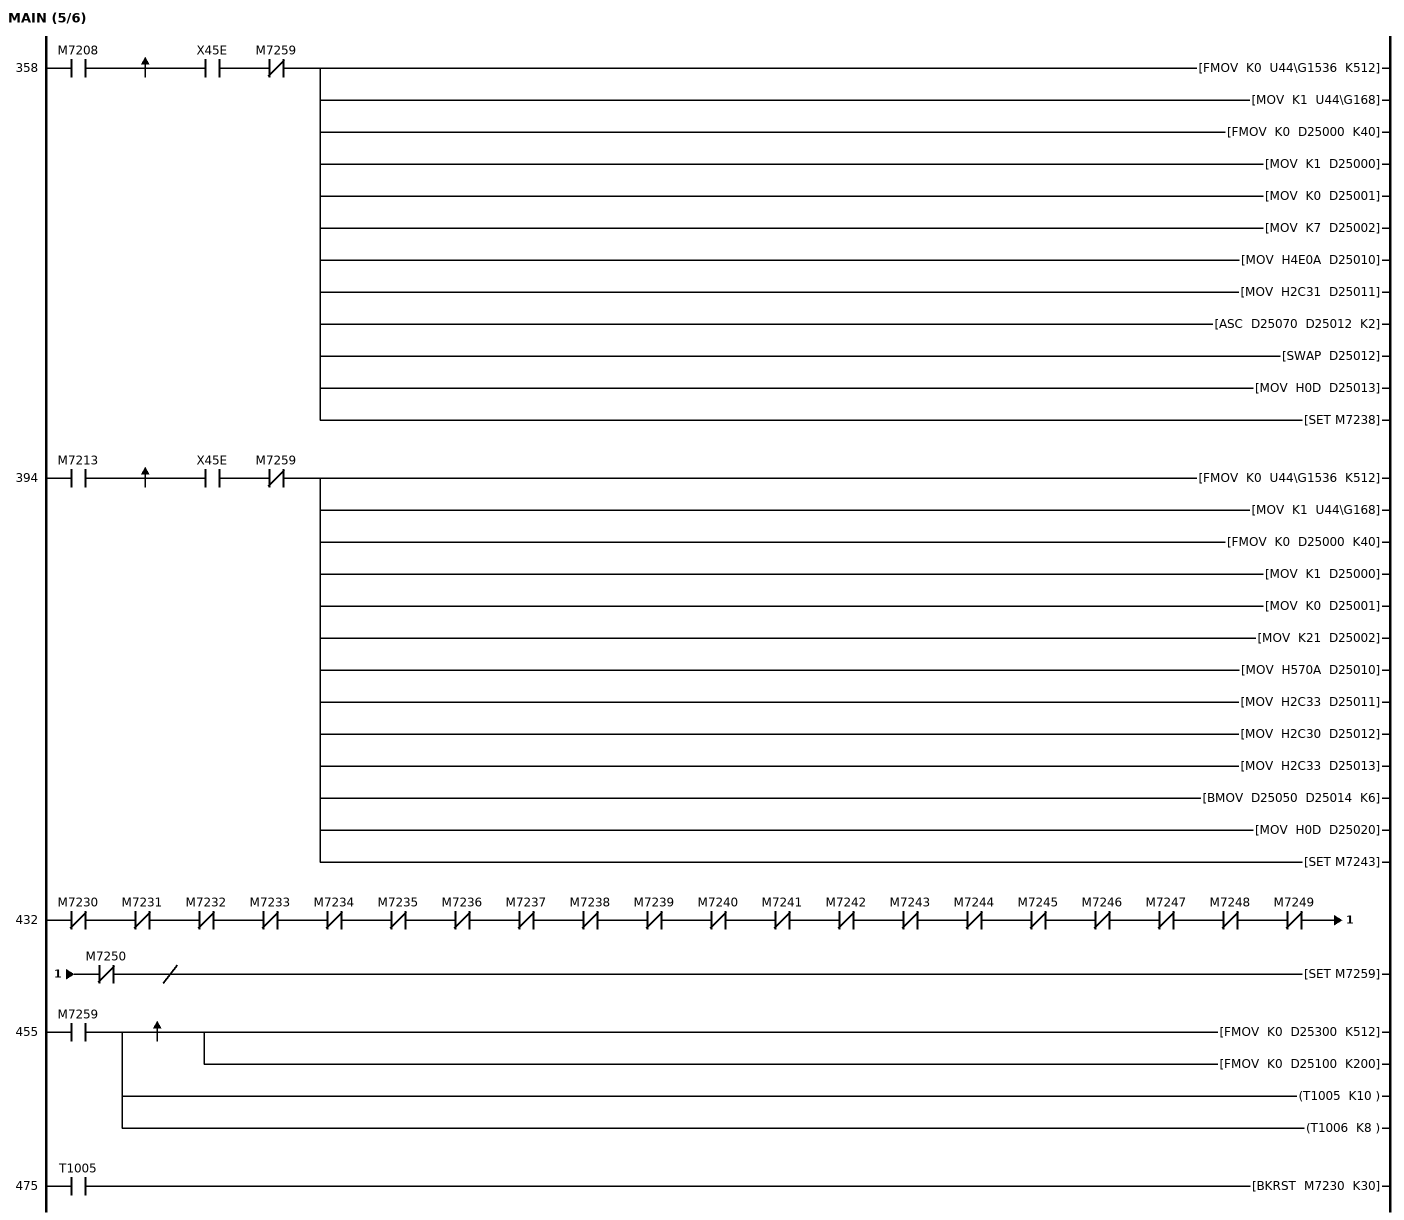
[picture p168: ladder of MAIN, rungs at steps 358 to 475]
358   LD      M7208
      MEP
      AND     X45E
      ANI     M7259
      FMOV    K0 U44\G1536 K512
      MOV     K1 U44\G168
      FMOV    K0 D25000 K40
      MOV     K1 D25000
      MOV     K0 D25001
      MOV     K7 D25002
      MOV     H4E0A D25010
      MOV     H2C31 D25011
      ASC     D25070 D25012 K2
      SWAP    D25012
      MOV     H0D D25013
      SET     M7238
394   LD      M7213
      MEP
      AND     X45E
      ANI     M7259
      FMOV    K0 U44\G1536 K512
      MOV     K1 U44\G168
      FMOV    K0 D25000 K40
      MOV     K1 D25000
      MOV     K0 D25001
      MOV     K21 D25002
      MOV     H570A D25010
      MOV     H2C33 D25011
      MOV     H2C30 D25012
      MOV     H2C33 D25013
      BMOV    D25050 D25014 K6
      MOV     H0D D25020
      SET     M7243
432   LDI     M7230
      ANI     M7231
      ANI     M7232
      ANI     M7233
      ANI     M7234
      ANI     M7235
      ANI     M7236
      ANI     M7237
      ANI     M7238
      ANI     M7239
      ANI     M7240
      ANI     M7241
      ANI     M7242
      ANI     M7243
      ANI     M7244
      ANI     M7245
      ANI     M7246
      ANI     M7247
      ANI     M7248
      ANI     M7249
      ANI     M7250
      INV
      SET     M7259
455   LD      M7259
      MPS
      MEP
      FMOV    K0 D25300 K512
      FMOV    K0 D25100 K200
      MPP
      OUT     T1005 K10
      OUT     T1006 K8
475   LD      T1005
      BKRST   M7230 K30
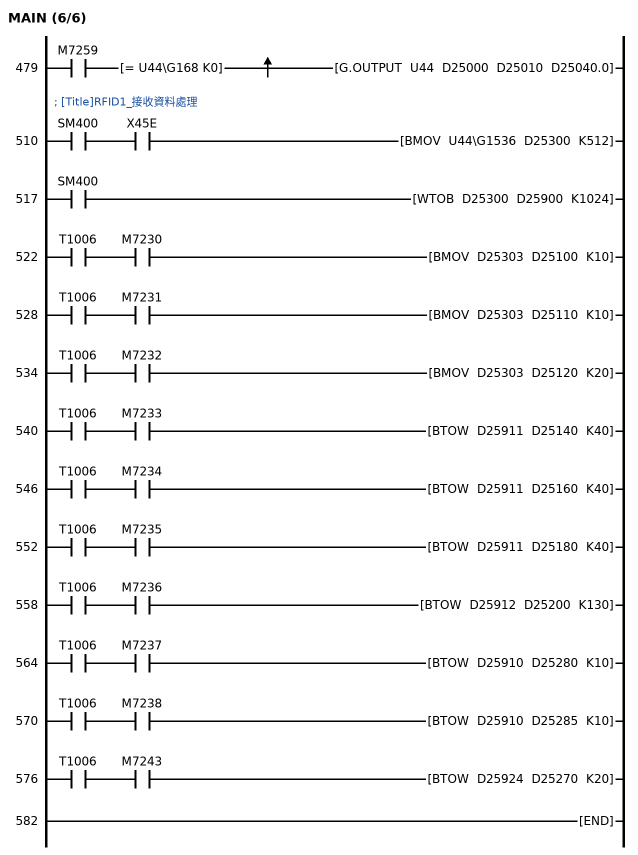
479   LD      M7259
      AND=    U44\G168 K0
      MEP
      G.OUTPUT U44 D25000 D25010 D25040.0
; [Title]RFID1_接收資料處理
510   LD      SM400
      AND     X45E
      BMOV    U44\G1536 D25300 K512
517   LD      SM400
      WTOB    D25300 D25900 K1024
522   LD      T1006
      AND     M7230
      BMOV    D25303 D25100 K10
528   LD      T1006
      AND     M7231
      BMOV    D25303 D25110 K10
534   LD      T1006
      AND     M7232
      BMOV    D25303 D25120 K20
540   LD      T1006
      AND     M7233
      BTOW    D25911 D25140 K40
546   LD      T1006
      AND     M7234
      BTOW    D25911 D25160 K40
552   LD      T1006
      AND     M7235
      BTOW    D25911 D25180 K40
558   LD      T1006
      AND     M7236
      BTOW    D25912 D25200 K130
564   LD      T1006
      AND     M7237
      BTOW    D25910 D25280 K10
570   LD      T1006
      AND     M7238
      BTOW    D25910 D25285 K10
576   LD      T1006
      AND     M7243
      BTOW    D25924 D25270 K20
582   END
END_PROGRAM

// device comments not shown above
X14  ; 下料旋臂長程中定點
X3D  ; 輸送機輸送馬達  INV41運轉
X3E  ; 中心機輸送馬達  INV42運轉
X31D  ; 30
X327  ; 40
X331  ; 50
X332  ; FR1-DO(31)
X333  ; FR1-DO(32)
X334  ; FR1-DO(33)
X335  ; FR1-DO(34)
X337  ; FR1-DO(36)
X338  ; FR1-DO(37)
X339  ; FR1-DO(38)
X33A  ; FR1-DO(39)
X33B  ; FR1-DO(40)
X33C  ; FR1-DO(41)
X33D  ; FR1-DO(42)
X33E  ; FR1-DO(43)
X33F  ; FR1-DO(44)
X340  ; FR1-DO(45)
X341  ; FR1-DO(46)
X342  ; FR1-DO(47)
X343  ; FR1-DO(48)
X344  ; FR1-DO(49)
X345  ; FR1-DO(50)
X346  ; FR1-DO(51)
X347  ; FR1-DO(52)
X348  ; FR1-DO(53)
X349  ; FR1-DO(54)
X34A  ; FR1-DO(55)
X34B  ; FR1-DO(56)
X34C  ; FR1-DO(57)
X34D  ; FR1-DO(58)
X34E  ; FR1-DO(59)
X34F  ; FR1-DO(60)
X350  ; FR1-DO(61)
X351  ; FR1-DO(62)
X352  ; FR1-DO(63)
X353  ; FR1-DO(64)
X354  ; FR1-DO(65)
X355  ; FR1-DO(66)
X356  ; FR1-DO(67)
X357  ; FR1-DO(68)
X358  ; FR1-DO(69)
X359  ; FR1-DO(70)
X35A  ; FR1-DO(71)
X35B  ; FR1-DO(72)
X35C  ; FR1-DO(73)
X35D  ; FR1-DO(74)
X35E  ; FR1-DO(75)
X35F  ; FR1-DO(76)
X360  ; FR1-DO(77)
X361  ; FR1-DO(78)
X362  ; FR1-DO(79)
X363  ; FR1-DO(80)
X364  ; FR1-DO(81)
X365  ; FR1-DO(82)
X366  ; FR1-DO(83)
X367  ; FR1-DO(84)
X368  ; FR1-DO(85)
X369  ; FR1-DO(86)
X36A  ; FR1-DO(87)
X36B  ; FR1-DO(88)
X36C  ; FR1-DO(89)
X36D  ; FR1-DO(90)
X36E  ; FR1-DO(91)
X36F  ; FR1-DO(92)
X370  ; FR1-DO(93)
X371  ; FR1-DO(94)
X372  ; FR1-DO(95)
X373  ; FR1-DO(96)
X374  ; FR1-DO(97)
X375  ; FR1-DO(98)
X376  ; FR1-DO(99)
X377  ; FR1-DO(100)
X378  ; FR1-DO(101)
X379  ; FR1-DO(102)
X37A  ; FR1-DO(103)
X37B  ; FR1-DO(104)
X37C  ; FR1-DO(105)
X37D  ; FR1-DO(106)
X37E  ; FR1-DO(107)
X37F  ; FR1-DO(108)
X0A03  ; Other station   DataLinkStatus
X0A21  ; Synchronization flag
X0A24  ; #1 AXIS M碼On
X0A25  ; #2 AXIS M碼On
X0A26  ; #3 AXIS M碼On
X0A27  ; #4 AXIS M碼On
X0A2A  ; #3 AXIS Error
X0A2B  ; #4 AXIS Error
X0A2E  ; #3 AXIS Busy
X0A2F  ; #4 AXIS Busy
X0A30  ; #1 AXIS 啟動完成
X0A32  ; #3 AXIS 啟動完成
X0A33  ; #4 AXIS 啟動完成
X0A35  ; #2 AXIS 定位完成
X0A36  ; #3 AXIS 定位完成
X0A37  ; #4 AXIS 定位完成
Y10C  ; @進料連線--取板中
Y31D  ; 30
Y327  ; 40
Y330  ; TR1-DI(31)
Y331  ; TR1-DI(32)-50
Y332  ; TR1-DI(33)
Y333  ; TR1-DI(34)-52
Y334  ; TR1-DI(35)
Y335  ; TR1-DI(36)
Y336  ; TR1-DI(37)-55
Y337  ; TR1-DI(38)
Y338  ; TR1-DI(39)
Y339  ; TR1-DI(40)
Y33A  ; TR1-DI(41)
Y33B  ; TR1-DI(42)
Y33C  ; TR1-DI(43)
Y33D  ; TR1-DI(44)
Y33E  ; TR1-DI(45)
Y33F  ; TR1-DI(46)
Y340  ; TR1-DI(47)
Y341  ; TR1-DI(48)
Y342  ; TR1-DI(49)
Y343  ; TR1-DI(50)
Y344  ; TR1-DI(51)
Y345  ; TR1-DI(52)
Y346  ; TR1-DI(53)
Y347  ; TR1-DI(54)
Y348  ; TR1-DI(55)
Y349  ; TR1-DI(56)
Y34A  ; TR1-DI(57)
Y34B  ; TR1-DI(58)
Y34C  ; TR1-DI(59)
Y34D  ; TR1-DI(60)
Y34E  ; TR1-DI(61)
Y34F  ; TR1-DI(62)
Y350  ; TR1-DI(63)
Y351  ; TR1-DI(64)
Y352  ; TR1-DI(65)
Y353  ; TR1-DI(66)
Y354  ; TR1-DI(67)
Y355  ; TR1-DI(68)
Y356  ; TR1-DI(69)
Y357  ; TR1-DI(70)
Y358  ; TR1-DI(71)
Y359  ; TR1-DI(72)
Y35A  ; TR1-DI(73)
Y35B  ; TR1-DI(74)
Y35C  ; TR1-DI(75)
Y35D  ; TR1-DI(76)
Y35E  ; TR1-DI(77)
Y35F  ; TR1-DI(78)
Y360  ; TR1-DI(79)
Y361  ; TR1-DI(80)
Y362  ; TR1-DI(81)
Y363  ; TR1-DI(82)
Y364  ; TR1-DI(83)
Y365  ; TR1-DI(84)
Y366  ; TR1-DI(85)
Y367  ; TR1-DI(86)
Y368  ; TR1-DI(87)
Y369  ; TR1-DI(88)
Y36A  ; TR1-DI(89)
Y36B  ; TR1-DI(90)
Y36C  ; TR1-DI(91)
Y36D  ; TR1-DI(92)
Y36E  ; TR1-DI(93)
Y36F  ; TR1-DI(94)
Y370  ; TR1-DI(95)
Y371  ; TR1-DI(96)
Y372  ; TR1-DI(97)
Y373  ; TR1-DI(98)
Y374  ; TR1-DI(99)
Y375  ; TR1-DI(100)
Y376  ; TR1-DI(101)
Y377  ; TR1-DI(102)
Y378  ; TR1-DI(103)
Y379  ; TR1-DI(104)
Y37A  ; TR1-DI(105)
Y37B  ; TR1-DI(106)
Y37C  ; TR1-DI(107)
Y37D  ; TR1-DI(108)
Y37E  ; TR1-DI(109)
Y37F  ; TR1-DI(110)
Y0A26  ; #3 AXIS Stop
Y0A27  ; #4 AXIS Stop
Y0A2C  ; #3 AXIS JOG+
Y0A2D  ; #3 AXIS JOG-
Y0A2E  ; #4 AXIS JOG+
Y0A2F  ; #4 AXIS JOG-
Y0A32  ; #3 AXIS Start
Y0A33  ; #4 AXIS Start
Y0A34  ; #1 AXIS 執行禁止
Y0A35  ; #2 AXIS 執行禁止
Y0A36  ; #3 AXIS 執行禁止
Y0A37  ; #4 AXIS 執行禁止
M70  ; 昇降上昇位置教導設定PB
M71  ; 昇降上等待位置教導設定PB
M73  ; 昇降下降位置教導設定PB
M76  ; 下料鼓風機自動
M79  ; 下料鼓風機手動
M190  ; 上料掉板後原點復歸
M191  ; 上料掉板後原點復歸STOP
M237  ; 上料夾爪可伸出KP
M332  ; 進料輸送停止
M333  ; 進料輸送減速KP
M514  ; 下料旋臂長程中定點
M552  ; 進料集塵鼓風機手動運轉
M553  ; 出料風車訊號
M554  ; 進出料集塵鼓風機自動運轉
M572  ; #13 風車啟動PB
M573  ; #14 風車啟動PB
M574  ; #15 風車啟動PB
M575  ; #16 風車啟動PB
M576  ; #17 風車啟動PB
M577  ; #18 風車啟動PB
M578  ; #19 風車啟動PB
M579  ; #20 風車啟動PB
M580  ; #21 風車啟動PB
M581  ; #22 風車啟動PB
M582  ; #23 風車啟動PB
M583  ; #24 風車啟動PB
M584  ; #25 風車啟動PB
M585  ; #26 風車啟動PB
M586  ; #27 風車啟動PB
M587  ; #28 風車啟動PB
M588  ; #29 風車啟動PB
M589  ; #30 風車啟動PB
M590  ; #31 風車啟動PB
M591  ; #32 風車啟動PB
M606  ; #13 電熱啟動PB
M607  ; #14 電熱啟動PB
M608  ; #15 電熱啟動PB
M609  ; #16 電熱啟動PB
M610  ; #17 電熱啟動PB
M611  ; #18 電熱啟動PB
M612  ; #19 電熱啟動PB
M613  ; #20 電熱啟動PB
M614  ; #21 電熱啟動PB
M615  ; #22 電熱啟動PB
M616  ; #23 電熱啟動PB
M617  ; #24 電熱啟動PB
M618  ; #25 電熱啟動PB
M619  ; #26 電熱啟動PB
M620  ; #27 電熱啟動PB
M621  ; #28 電熱啟動PB
M622  ; #29 電熱啟動PB
M623  ; #30 電熱啟動PB
M624  ; #31 電熱啟動PB
M625  ; #32 電熱啟動PB
M639  ; 排氣風壓檢知異常警報
M659  ; 排氣風壓檢知異常警報PLS
M732  ; #13 風車訊號
M733  ; #14 風車訊號
M734  ; #15 風車訊號
M735  ; #16 風車訊號
M736  ; #17 風車訊號
M737  ; #18 風車訊號
M738  ; #19 風車訊號
M739  ; #20 風車訊號
M740  ; #21 風車訊號
M741  ; #22 風車訊號
M742  ; #23 風車訊號
M743  ; #24 風車訊號
M744  ; #25 風車訊號
M745  ; #26 風車訊號
M746  ; #27 風車訊號
M747  ; #28 風車訊號
M748  ; #29 風車訊號
M749  ; #30 風車訊號
M750  ; #31 風車訊號
M751  ; #32 風車訊號
M792  ; #13 電熱訊號
M793  ; #14 電熱訊號
M794  ; #15 電熱訊號
M795  ; #16 電熱訊號
M796  ; #17 電熱訊號
M797  ; #18 電熱訊號
M798  ; #19 電熱訊號
M799  ; #20 電熱訊號
M800  ; #21 電熱訊號
M801  ; #22 電熱訊號
M802  ; #23 電熱訊號
M803  ; #24 電熱訊號
M804  ; #25 電熱訊號
M805  ; #26 電熱訊號
M806  ; #27 電熱訊號
M807  ; #28 電熱訊號
M808  ; #29 電熱訊號
M809  ; #30 電熱訊號
M810  ; #31 電熱訊號
M811  ; #32 電熱訊號
M832  ; #13 溫度到達KP
M833  ; #14 溫度到達KP
M834  ; #15 溫度到達KP
M835  ; #16 溫度到達KP
M836  ; #17 溫度到達KP
M837  ; #18 溫度到達KP
M838  ; #19 溫度到達KP
M839  ; #20 溫度到達KP
M840  ; #21 溫度到達KP
M841  ; #22 溫度到達KP
M842  ; #23 溫度到達KP
M843  ; #24 溫度到達KP
M844  ; #25 溫度到達KP
M845  ; #26 溫度到達KP
M846  ; #27 溫度到達KP
M847  ; #28 溫度到達KP
M848  ; #29 溫度到達KP
M849  ; #30 溫度到達KP
M850  ; #31 溫度到達KP
M851  ; #32 溫度到達KP
M1304  ; 進料段無板
M1305  ; 進料定位有板
M1412  ; #13 風車啟動PLS
M1413  ; #14 風車啟動PLS
M1414  ; #15 風車啟動PLS
M1415  ; #16 風車啟動PLS
M1416  ; #17 風車啟動PLS
M1417  ; #18 風車啟動PLS
M1418  ; #19 風車啟動PLS
M1419  ; #20 風車啟動PLS
M1420  ; #21 風車啟動PLS
M1421  ; #22 風車啟動PLS
M1422  ; #23 風車啟動PLS
M1423  ; #24 風車啟動PLS
M1424  ; #25 風車啟動PLS
M1425  ; #26 風車啟動PLS
M1426  ; #27 風車啟動PLS
M1427  ; #28 風車啟動PLS
M1428  ; #29 風車啟動PLS
M1429  ; #30 風車啟動PLS
M1430  ; #31 風車啟動PLS
M1431  ; #32 風車啟動PLS
M1452  ; #13 電熱啟動PLS
M1453  ; #14 電熱啟動PLS
M1454  ; #15 電熱啟動PLS
M1455  ; #16 電熱啟動PLS
M1456  ; #17 電熱啟動PLS
M1457  ; #18 電熱啟動PLS
M1458  ; #19 電熱啟動PLS
M1459  ; #20 電熱啟動PLS
M1460  ; #21 電熱啟動PLS
M1461  ; #22 電熱啟動PLS
M1462  ; #23 電熱啟動PLS
M1463  ; #24 電熱啟動PLS
M1464  ; #25 電熱啟動PLS
M1465  ; #26 電熱啟動PLS
M1466  ; #27 電熱啟動PLS
M1467  ; #28 電熱啟動PLS
M1468  ; #29 電熱啟動PLS
M1469  ; #30 電熱啟動PLS
M1470  ; #31 電熱啟動PLS
M1471  ; #32 電熱啟動PLS
M1481  ; 進料風車2啟動PLS
M1482  ; 進料風車3啟動PLS
M1491  ; 出料風車2啟動PLS
M1492  ; 出料風車3啟動PLS
M1512  ; #13 電熱停止PLS
M1513  ; #14 電熱停止PLS
M1514  ; #15 電熱停止PLS
M1515  ; #16 電熱停止PLS
M1516  ; #17 電熱停止PLS
M1517  ; #18 電熱停止PLS
M1518  ; #19 電熱停止PLS
M1519  ; #20 電熱停止PLS
M1520  ; #21 電熱停止PLS
M1521  ; #22 電熱停止PLS
M1522  ; #23 電熱停止PLS
M1523  ; #24 電熱停止PLS
M1524  ; #25 電熱停止PLS
M1525  ; #26 電熱停止PLS
M1526  ; #27 電熱停止PLS
M1527  ; #28 電熱停止PLS
M1528  ; #29 電熱停止PLS
M1529  ; #30 電熱停止PLS
M1530  ; #31 電熱停止PLS
M1531  ; #32 電熱停止PLS
M1552  ; #13 風車停止PLS
M1553  ; #14 風車停止PLS
M1554  ; #15 風車停止PLS
M1555  ; #16 風車停止PLS
M1556  ; #17 風車停止PLS
M1557  ; #18 風車停止PLS
M1558  ; #19 風車停止PLS
M1559  ; #20 風車停止PLS
M1560  ; #21 風車停止PLS
M1561  ; #22 風車停止PLS
M1562  ; #23 風車停止PLS
M1563  ; #24 風車停止PLS
M1564  ; #25 風車停止PLS
M1565  ; #26 風車停止PLS
M1566  ; #27 風車停止PLS
M1567  ; #28 風車停止PLS
M1568  ; #29 風車停止PLS
M1569  ; #30 風車停止PLS
M1570  ; #31 風車停止PLS
M1571  ; #32 風車停止PLS
M1581  ; 進料風車2停止PLS
M1582  ; 進料風車3停止PLS
M1591  ; 出料風車2停止PLS
M1592  ; 出料風車3停止PLS
M2003  ; Axis01  STOP
M2008  ; Axis01  伺服啟動
M2011  ; Axis01  速度轉換位置
M2012  ; Axis01  命令近點
M2013  ; Axis01  歸零要求
M2014  ; Axis01  歸零完成
M2018  ; Axis01  伺服啟動
M2019  ; Axis01  伺服啟動異常
M2020  ; Axis01  移載異常
M2021  ; Axis01  移載警告
M2022  ; Axis01  寸動可運轉
M2023  ; Axis01  命令可運轉
M2024  ; Axis01  歸零完成PLS
M2025  ; Axis01  DO HOME
M2026  ; Axis01  啟動完成
M2027  ; Axis01  DO HOMO 完成
M2028  ; Axis01  要求回原點
M2029  ; Axis01  己回原點
M2030  ; Axis01  移載位置01
M2031  ; Axis01  移載位置02
M2032  ; Axis01  移載位置03
M2033  ; Axis01  移載位置04
M2034  ; Axis01  移載位置05
M2035  ; Axis01  移載位置06
M2036  ; Axis01  移載位置07
M2037  ; Axis01  移載位置08
M2038  ; Axis01  移載位置09
M2039  ; Axis01  移載位置10
M2040  ; Axis01  位置01  訊號
M2041  ; Axis01  位置02  訊號
M2042  ; Axis01  位置03  訊號
M2043  ; Axis01  位置04  訊號
M2044  ; Axis01  位置05  訊號
M2045  ; Axis01  位置06  訊號
M2046  ; Axis01  位置07  訊號
M2047  ; Axis01  位置08  訊號
M2048  ; Axis01  位置09  訊號
M2049  ; Axis01  位置10  訊號
M2050  ; Axis01  READY ON
M2051  ; Axis01  Servo ON
M2054  ; Axis01  Zero point pass
M2055  ; Axis01  In-position
M2056  ; Axis01  Zero speed
M2057  ; Axis01  Torque limit
M2063  ; Axis01  Servo alarm
M2064  ; Axis01  Servo warning
M2070  ; Axis01  速度控制
M2071  ; Axis01  速度轉換位置
M2072  ; Axis01  命令近點
M2073  ; Axis01  歸零要求
M2074  ; Axis01  歸零完成
M2082  ; Axis01  M code ON
M2083  ; Axis01  Error detection
M2084  ; Axis01  Start complete
M2085  ; Axis01  Positioning complete
M2103  ; Axis02  STOP
M2108  ; Axis02  伺服啟動
M2111  ; Axis02  速度轉換位置
M2112  ; Axis02  命令近點
M2113  ; Axis02  歸零要求
M2114  ; Axis02  歸零完成
M2118  ; Axis02  伺服啟動
M2119  ; Axis02  伺服啟動異常
M2120  ; Axis02  移載異常
M2121  ; Axis02  移載警告
M2122  ; Axis02  寸動可運轉
M2123  ; Axis02  命令可運轉
M2124  ; Axis02  歸零完成PLS
M2125  ; Axis02  DO HOME
M2126  ; Axis02  啟動完成
M2127  ; Axis02  DO HOMO 完成
M2128  ; Axis02  要求回原點
M2129  ; Axis02  己回原點
M2130  ; Axis02  移載位置01
M2131  ; Axis02  移載位置02
M2132  ; Axis02  移載位置03
M2133  ; Axis02  移載位置04
M2134  ; Axis02  移載位置05
M2135  ; Axis02  移載位置06
M2136  ; Axis02  移載位置07
M2137  ; Axis02  移載位置08
M2138  ; Axis02  移載位置09
M2139  ; Axis02  移載位置10
M2140  ; Axis02  位置01  訊號
M2141  ; Axis02  位置02  訊號
M2142  ; Axis02  位置03  訊號
M2143  ; Axis02  位置04  訊號
M2144  ; Axis02  位置05  訊號
M2145  ; Axis02  位置06  訊號
M2146  ; Axis02  位置07  訊號
M2147  ; Axis02  位置08  訊號
M2148  ; Axis02  位置09  訊號
M2149  ; Axis02  位置10  訊號
M2150  ; Axis02  READY ON
M2151  ; Axis02  Servo ON
M2154  ; Axis02  Zero point pass
M2155  ; Axis02  In-position
M2156  ; Axis02  Zero speed
M2157  ; Axis02  Torque limit
M2163  ; Axis02  Servo alarm
M2164  ; Axis02  Servo warning
M2170  ; Axis02  速度控制
M2171  ; Axis02  速度轉換位置
M2172  ; Axis02  命令近點
M2173  ; Axis02  歸零要求
M2174  ; Axis02  歸零完成
M2182  ; Axis02  M code ON
M2183  ; Axis02  Error detection
M2184  ; Axis02  Start complete
M2185  ; Axis02  Positioning complete
M2707  ; A6Ini_軟板到位
M2718  ; A6Ini_初始化失敗
M2721  ; A6Auto_檢查有無板
M2722  ; A6Auto_檢查無板
M2723  ; A6Auto_平台下降
M2724  ; A6Auto_前後擋退開
M2725  ; A6Auto_左右擋退開
M2726  ; A6Auto_左右壓板退開
M2727  ; A6Auto_C/V收板請求
M2728  ; A6Auto_C/V收板Busy
M2729  ; A6Auto_C/V收板到位
M2859  ; 中心拍板伺服寸動往內PB燈
M2860  ; 中心拍板伺服寸動往外PB燈
M2890  ; 中心拍板伺服設定位置KP
M2900  ; 中心拍板伺服內極限燈
M2901  ; 中心拍板設定位置燈
M2903  ; 中心拍板夾爪原點位置燈
M2904  ; 中心拍板夾爪伺服原點燈
M2905  ; 中心拍板夾爪伺服外極限燈
M2910  ; 中心拍板設定位置
M2912  ; 中心拍板原點位置
M2920  ; 中心拍板設定位置
M3090  ; 拍板馬達伺服原點訊號PLS1
M3156  ; 拍板馬達至原點PB燈
M3158  ; 拍板馬達原點復歸PB燈
M3188  ; 拍板馬達伺服原點復歸
M3258  ; 拍板馬達伺服原點位置自動
M3319  ; 拍板馬達伺服原點復歸OK
M3358  ; 拍板馬達伺服原點位置手動
M3385  ; 拍板馬達伺服可動作
M3390  ; 拍板馬達設定位置KP
M3393  ; 拍板馬達原點位置KP
M3394  ; 拍板馬達伺服原點復歸KP
M3395  ; 拍板馬達伺服開機原點復歸KP
M3400  ; 拍板馬達伺服內極限燈
M3403  ; 拍板馬達原點位置燈
M3405  ; 拍板馬達伺服外極限燈
M3410  ; 拍板馬達設定位置
M3412  ; 拍板馬達原點位置
M3422  ; 拍板馬達原點位置
M4678  ; 拍板馬達伺服異常
M4704  ; 生產片數到達
M4713  ; 拍板馬達伺服運轉逾時異常
M4716  ; 拍板馬達伺服內極限
M4717  ; 拍板馬達伺服外極限
M4917  ; 刪除配方名稱
M4921  ; 出口計數
M4922  ; 爐內限制異常
M4923  ; 出口計數
M4925  ; 卡板不警報
M4930  ; 點燈運轉KP
M4931  ; 點燈停止
M4932  ; 上位下啟動訊號
M4933  ; PP_SELECT點燈用保持
M4937  ; 上位要儲存配方
M4950  ; 點燈中請稍待指示
M4951  ; 熄點燈冷卻中請稍待指示
M4953  ; 熄燈OK狀態
M4956  ; 輸送機停止熄燈
M4990  ; 密碼ENT
M4992  ; 密碼ENT Keep
M4993  ; 參數設定取消PB
M4994  ; 參數設定取消PLS
M4996  ; 離線測試用
M5034  ; 輸送運轉未加熱完成
M5101  ; 三色紅燈
M5102  ; 三色綠燈
M5215  ; Barcod啟動固定式完成
M5217  ; 門,(1)(2),PPID,配方名稱比對不對
M5314  ; 配方刪除
M5315  ; 配方儲存
M5316  ; 呼叫Q的配方
M5317  ; 比對配方用
M5318  ; 自動
M5319  ; 手動
M5321  ; 自動啟動
M5325  ; 對話視窗關閉
M5326  ; 配方新增
M5327  ; 配方修改
M5328  ; 配方刪除
M5329  ; 機構異常警報
M5347  ; 配方Barcode掃描
M5348  ; 工單輸入
M5349  ; Barcod啟動固定式
M5350  ; Bey Pass PB
M5351  ; 自動PB
M5352  ; 連線開放OP控制
M5353  ; 確認(101頁)人機SET
M5354  ; 確認(102頁)人機SET
M6059  ; Host刪除配方
M6060  ; Host刪除配方完成
M6140  ; 要求上位回讀工單板號右爐
M6141  ; 要求上位回讀工單右爐
M6231  ; 上位要儲存配方
M6300  ; 緊急停止開關異常
M6301  ; 逆相繼電器異常
M6302  ; 入口卡板異常
M6303  ; 出口卡板異常
M6304  ; UV門防止打開開關異常
M6305  ; 上排風風車過載
M6306  ; 下排風風車過載
M6307  ; 安定器冷卻風扇過載
M6308  ; 第一燈溫度異常
M6309  ; 下燈1點燈異常
M6310  ; 下燈2點燈異常
M6311  ; 上燈1點燈異常
M6312  ; 上燈2點燈異常
M6313  ; 變頻機異常
M6314  ; 出料連線異常
M6315  ; 爐內限制數量異常
M6316  ; PLC Low Battery
M6317  ; 進氣冷卻風扇過載
M6318  ; 燈箱冷卻風扇過載
M6319  ; 輸送運轉未點燈警報
M6320  ; 點燈中輸送停止未運轉
M6321  ; 板子有進沒出m231沒滅
M6322  ; 輸送馬達過載異常
M6323  ; 網偏前警報
M6324  ; 網偏後警報
M6325  ; 燈箱冷卻風扇過載
M6326  ; 進氣冷卻風扇過載
M6327  ; 網偏警報熄燈計時
M6328  ; 第二燈溫度異常
M6330  ; UV點燈後30秒不可選擇提示
M6331  ; 下燈1管保養時間到達
M6332  ; 下燈2管保養時間到達
M6333  ; 上燈1管保養時間到達
M6334  ; 上燈2管保養時間到達
M6335  ; 滾輪保養時間到達
M6336  ; 輸送馬達過載異常
M6339  ; 節能省電啟動
M6340  ; 出口卡板異常
M6344  ; 安全門開啟時熄燈選擇    (on熄燈)
M6345  ; 卡板熄燈
M6349  ; 下燈1   點燈失敗
M6350  ; 下燈2   點燈失敗
M6351  ; 上燈1   點燈失敗
M6352  ; 上燈2   點燈失敗
M6607  ; Host刪除配方自保持
M6608  ; Host刪除配方自清除保持
M6610  ; 比對M700~M715都等於零
M6611  ; 比對M716~M731都等於零
M6854  ; 機台再IDEL
M6999  ; 三色綠燈
M7001  ; 三色紅燈
M7999  ; 暫時不開
D10  ; 靜置段風車
D11  ; 冷卻段風車
D13  ; 風車啟動數
D14  ; 加熱啟動數量
D22  ; 昇降伺服設定參數
D23  ; 昇降伺服異常碼
D24  ; 昇降伺服異常碼
D35  ; 年*10000
D37  ; 月*100
D39  ; 人機時間年月日
D41  ; 進料輸送停止時間延遲
D75  ; 加熱段長度W2
D78  ; 板架距離W2
D150  ; 人機參數密碼
D207  ; 取板基準點板長(0.1mm)
D220  ; 上料手臂取板位置換算
D221  ; 上料手臂取板位置暫存
D222  ; 上料手臂取板位置暫存
D249  ; 上料手臂夾爪現在位置換算板寬
D251  ; 上料手臂夾爪現在位置
D253  ; 上料手臂夾爪伺服現在速度
D261  ; 上料手臂夾爪運轉速度設定
D263  ; 上料手臂夾爪JOG速度值
D265  ; 上料手臂夾爪設定位置設定值
D267  ; 上料手臂夾爪原點位置設定值
D297  ; 總生產量Hi
D301  ; 本班產量履歷2
D302  ; 本班產量履歷3
D303  ; 本班產量履歷4
D304  ; 本班產量履歷5
D305  ; 本班產量履歷6
D306  ; 本班產量履歷7
D307  ; 本班產量履歷8
D308  ; 本班產量履歷9
D309  ; 本班產量履歷10
D310  ; 本班產量履歷11
D311  ; 本班產量履歷12
D312  ; 本班產量履歷13
D313  ; 本班產量履歷14
D314  ; 本班產量履歷15
D315  ; 本班產量履歷16
D316  ; 本班產量履歷17
D317  ; 本班產量履歷18
D318  ; 本班產量履歷19
D319  ; 本班產量履歷20
D320  ; 本班產量履歷21
D321  ; 本班產量履歷22
D322  ; 本班產量履歷23
D323  ; 本班產量履歷24
D324  ; 本班產量履歷25
D331  ; 現在時間時分2
D332  ; 現在時間時分3
D333  ; 現在時間時分4
D334  ; 現在時間時分5
D335  ; 現在時間時分6
D336  ; 現在時間時分7
D337  ; 現在時間時分8
D338  ; 現在時間時分9
D339  ; 現在時間時分10
D340  ; 現在時間時分11
D341  ; 現在時間時分12
D342  ; 現在時間時分13
D343  ; 現在時間時分14
D344  ; 現在時間時分15
D345  ; 現在時間時分16
D346  ; 現在時間時分17
D347  ; 現在時間時分18
D348  ; 現在時間時分19
D349  ; 現在時間時分20
D350  ; 現在時間時分21
D351  ; 現在時間時分22
D352  ; 現在時間時分23
D353  ; 現在時間時分24
D354  ; 現在時間時分25
D373  ; 動畫(PCB板出料現在位置)W2
D374  ; 動畫(PCB板出料現在位置)W3
D375  ; 動畫(PCB板出料現在位置)W4
D381  ; 動畫(長程氣缸上升現在位置)W2
D382  ; 動畫(長程氣缸上升現在位置)W3
D383  ; 動畫(長程氣缸上升現在位置)W4
D385  ; 動畫(旋臂水平現在位置)W2
D386  ; 動畫(旋臂水平現在位置)W3
D387  ; 動畫(旋臂水平現在位置)W4
D395  ; 月保養時間現在值
D397  ; 季保養時間現在值
D399  ; 年保養時間現在值
D400  ; PLC=>SV1
D401  ; PLC=>SV2
D402  ; PLC=>SV3
D403  ; PLC=>SV4
D404  ; PLC=>SV5
D405  ; PLC=>SV6
D406  ; PLC=>SV7
D407  ; PLC=>SV8
D408  ; PLC=>SV9
D409  ; PLC=>SV10
D420  ; PV1=>PLC
D421  ; PV2=>PLC
D422  ; PV3=>PLC
D423  ; PV4=>PLC
D424  ; PV5=>PLC
D425  ; PV6=>PLC
D426  ; PV7=>PLC
D427  ; PV8=>PLC
D428  ; PV9=>PLC
D429  ; PV10=>PLC
D440  ; SV1=>PLC
D441  ; SV2=>PLC
D442  ; SV3=>PLC
D443  ; SV4=>PLC
D444  ; SV5=>PLC
D445  ; SV6=>PLC
D446  ; SV7=>PLC
D447  ; SV8=>PLC
D448  ; SV9=>PLC
D449  ; SV10=>PLC
D473  ; 動畫(前一次旋臂水平時間)W2
D477  ; 動畫(前一次旋臂垂直時間)W2
D481  ; 動畫(前一次長程氣缸上升時間)W2
D485  ; 動畫(前一次長程氣缸下降時間)W2
D487  ; 動畫(長程氣缸下降時間X10)W2
D493  ; 動畫(前一次PCB板出料時間)W2
D495  ; 動畫(PCB板出料時間X10)W2
D497  ; 動畫(長程氣缸下降現在位置)W2
D498  ; 動畫(長程氣缸下降現在位置)W3
D499  ; 動畫(長程氣缸下降現在位置)W4
D507  ; 動畫(旋臂垂直現在位置)W2
D508  ; 動畫(旋臂垂直現在位置)W3
D509  ; 動畫(旋臂垂直現在位置)W4
D511  ; 動畫(旋臂垂直時間X10)W2
D548  ; 中心拍板現在位置換算板寬
D549  ; 中心拍板現在位置換算板寬
D551  ; 中心拍板夾爪現在位置
D553  ; 中心拍板夾爪伺服現在速度
D554  ; 中心拍板伺服異常碼
D561  ; 中心拍板運轉速度設定
D563  ; 中心拍板JOG速度值
D564  ; 中心拍板設定位置設定值
D565  ; 中心拍板設定位置設定值
D567  ; 中心拍板原點位置設定值
D641  ; 烘烤時間SEC
D701  ; 月保養時數
D711  ; 季保養時數
D721  ; 年保養時數
D809  ; 排氣風壓檢知異常警報
D859  ; 排氣風壓檢知異常警報暫存
D1001  ; 系統時間年月日00
D1002  ; 系統時間年月日01
D1003  ; 系統時間年月日01
D1004  ; 系統時間年月日02
D1005  ; 系統時間年月日02
D1006  ; 系統時間年月日03
D1007  ; 系統時間年月日03
D1008  ; 系統時間年月日04
D1009  ; 系統時間年月日04
D1010  ; 系統時間年月日05
D1011  ; 系統時間年月日05
D1012  ; 系統時間年月日06
D1013  ; 系統時間年月日06
D1014  ; 系統時間年月日07
D1015  ; 系統時間年月日07
D1016  ; 系統時間年月日08
D1017  ; 系統時間年月日08
D1018  ; 系統時間年月日09
D1019  ; 系統時間年月日09
D1020  ; 系統時間年月日10
D1021  ; 系統時間年月日10
D1022  ; 系統時間年月日11
D1023  ; 系統時間年月日11
D1024  ; 系統時間年月日12
D1025  ; 系統時間年月日12
D1026  ; 系統時間年月日13
D1027  ; 系統時間年月日13
D1028  ; 系統時間年月日14
D1029  ; 系統時間年月日14
D1030  ; 系統時間年月日15
D1031  ; 系統時間年月日15
D1032  ; 系統時間年月日16
D1033  ; 系統時間年月日16
D1034  ; 系統時間年月日17
D1035  ; 系統時間年月日17
D1036  ; 系統時間年月日18
D1037  ; 系統時間年月日18
D1038  ; 系統時間年月日19
D1039  ; 系統時間年月日19
D1040  ; 系統時間年月日20
D1041  ; 系統時間年月日20
D1042  ; 系統時間年月日21
D1043  ; 系統時間年月日21
D1044  ; 系統時間年月日22
D1045  ; 系統時間年月日22
D1046  ; 系統時間年月日23
D1047  ; 系統時間年月日23
D1048  ; 系統時間年月日24
D1049  ; 系統時間年月日24
D2000  ; TR1 ROBOT取板點(補償)X
D2001  ; TR1 ROBOT取板點(補償)Y
D2002  ; TR1 ROBOT取板點(補償)Z
D2008  ; TR1 ROBOT放板點(補償)X
D2009  ; TR1 ROBOT放板點(補償)Y
D2010  ; TR1 ROBOT放板點(補償)Z
D2101  ; TR1(R31)手臂取板點(補償)X
D2102  ; TR1(R32)手臂取板點(補償)Y
D2103  ; TR1(R33)手臂取板點(補償)Z
D2104  ; TR1(R34)手臂取板點(補償)角度
D2105  ; TR1(R35)手臂放板點(補償)X
D2106  ; TR1(R36)手臂放板點(補償)Y
D2107  ; TR1(R37)手臂放板點(補償)Z
D2109  ; TR1(R39)板長尺寸偏差量(0.1mm)
D2110  ; TR1(R40)
D2111  ; TR1(R41)
D2112  ; TR1(R42)
D2113  ; TR1(R43)
D2114  ; TR1(R44)
D2115  ; TR1(R45)
D2509  ; 板長尺寸偏差量計算(0.1mm)
D3243  ; 拍板原點位置板寬暫存(0.1mm)
D3250  ; 拍板馬達現在位置
D3252  ; 拍板馬達現在速度
D3260  ; 拍板馬達運轉速度設定
D3262  ; 拍板馬達JOG速度值
D3266  ; 拍板馬達原點位置設定值
D3302  ; 當前使用配方RecipeID#04/03
D3303  ; 當前使用配方RecipeID#06/05
D3304  ; 當前使用配方RecipeID#08/07
D3305  ; 當前使用配方RecipeID#10/09
D3306  ; 當前使用配方RecipeID#12/11
D3307  ; 當前使用配方RecipeID#14/13
D3308  ; 當前使用配方RecipeID#16/15
D3309  ; 當前使用配方RecipeID#18/17
D3310  ; 當前使用配方RecipeID#20/19
D3311  ; 當前使用配方RecipeID#22/21
D3312  ; 當前使用配方RecipeID#24/23
D3313  ; 當前使用配方RecipeID#26/25
D3314  ; 當前使用配方RecipeID#28/27
D3315  ; 當前使用配方RecipeID#30/29
D3316  ; 當前使用配方RecipeID#32/31
D3317  ; 當前使用配方RecipeID#34/33
D3318  ; 當前使用配方RecipeID#36/35
D3319  ; 當前使用配方RecipeID#38/37
D3320  ; 當前使用配方RecipeID#40/39
D3322  ; 當前使用配方第02槽電熱設定
D3323  ; 當前使用配方第03槽電熱設定
D3324  ; 當前使用配方第04槽電熱設定
D3325  ; 當前使用配方第05槽電熱設定
D3326  ; 當前使用配方第06槽電熱設定
D3327  ; 當前使用配方第07槽電熱設定
D3328  ; 當前使用配方第08槽電熱設定
D3329  ; 當前使用配方第09槽電熱設定
D3330  ; 當前使用配方第10槽電熱設定
D3331  ; 當前使用配方第11槽電熱設定
D3332  ; 當前使用配方第12槽電熱設定
D3390  ; HMI-編輯RecipeID#22/21
D3391  ; HMI-編輯RecipeID#24/23
D3392  ; HMI-編輯RecipeID#26/25
D3393  ; HMI-編輯RecipeID#28/27
D3394  ; HMI-編輯RecipeID#30/29
D3395  ; HMI-編輯RecipeID#32/31
D3396  ; HMI-編輯RecipeID#34/33
D3397  ; HMI-編輯RecipeID#36/35
D3398  ; HMI-編輯RecipeID#38/37
D3399  ; HMI-編輯RecipeID#40/39
D3420  ; HMI-編輯爐內烘烤時間計算-2(秒)
D3422  ; HMI-編輯爐內烘烤時間計算-2(分)
D4940  ; SP.SOC OPEN指令控制數據
D4944  ; SP.SOC SND指令結束元件
D4950  ; SP.SOC  SND指令控制數據
D4952  ; SP.SOC  RCV指令控制數據
D4954  ; SP.SOC  CLOSE指令控制數據
D5003  ; GP->ATMA_ROBOT準備取板
D5004  ; GP->ATMA_ROBOT動作完成
